PROGRAM pouStation2
VAR
	stationMode: FB_Mode;
	tCalcNumberOfPages: REAL;
	ceil: REAL;
	PartBuild: FB_PartBuild;
	retvall: UDINT;
	// TODO
	tPartPresent: BOOL;
END_VAR

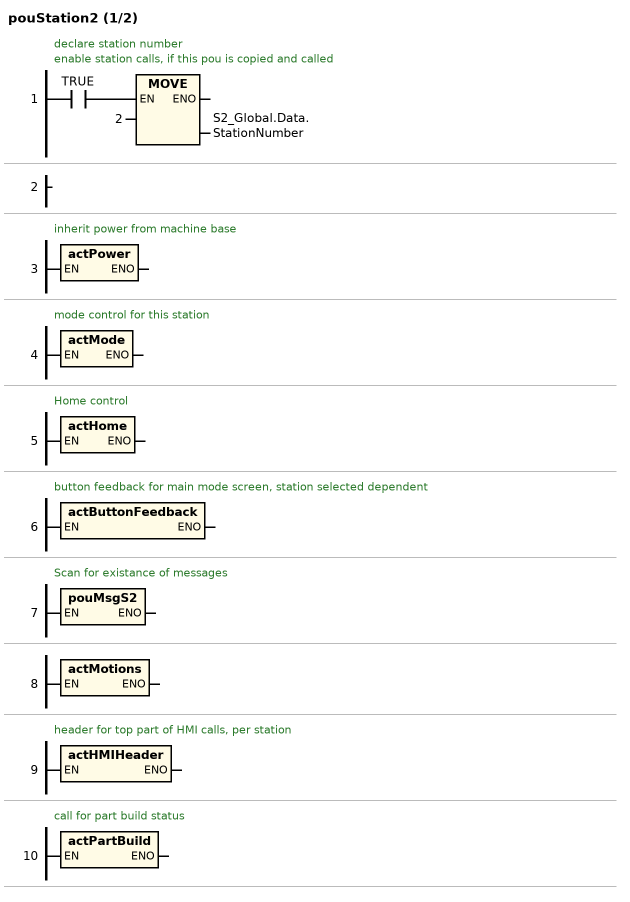
// NETWORK 1
// declare station number
// enable station calls, if this pou is copied and called
S2_Global.Data.StationNumber := 2;

// NETWORK 2

// NETWORK 3
// inherit power from machine base
actPower();

// NETWORK 4
// mode control for this station
actMode();

// NETWORK 5
// Home control
actHome();

// NETWORK 6
// button feedback for main mode screen, station selected dependent
actButtonFeedback();

// NETWORK 7
// Scan for existance of messages
pouMsgS2();

// NETWORK 8
actMotions();

// NETWORK 9
// header for top part of HMI calls, per station
actHMIHeader();

// NETWORK 10
// call for part build status
actPartBuild();

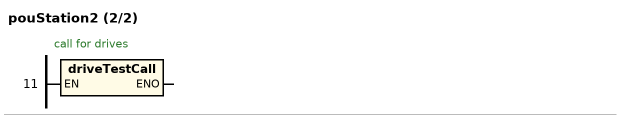
// NETWORK 11
// call for drives
driveTestCall();

ACTION actButtonFeedback:
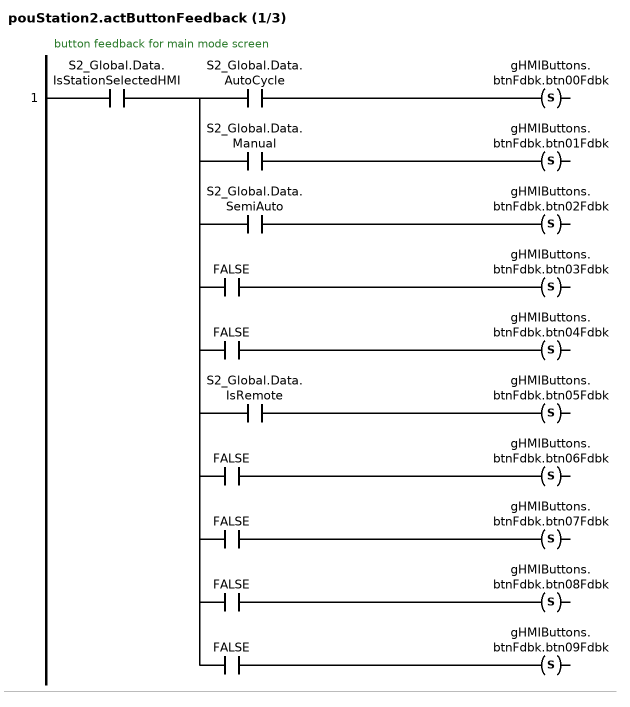
// NETWORK 1
// button feedback for main mode screen
gHMIButtons.btnFdbk.btn00Fdbk S= S2_Global.Data.IsStationSelectedHMI AND S2_Global.Data.AutoCycle;
gHMIButtons.btnFdbk.btn01Fdbk S= S2_Global.Data.IsStationSelectedHMI AND S2_Global.Data.Manual;
gHMIButtons.btnFdbk.btn02Fdbk S= S2_Global.Data.IsStationSelectedHMI AND S2_Global.Data.SemiAuto;
gHMIButtons.btnFdbk.btn03Fdbk S= S2_Global.Data.IsStationSelectedHMI AND FALSE;
gHMIButtons.btnFdbk.btn04Fdbk S= S2_Global.Data.IsStationSelectedHMI AND FALSE;
gHMIButtons.btnFdbk.btn05Fdbk S= S2_Global.Data.IsStationSelectedHMI AND S2_Global.Data.IsRemote;
gHMIButtons.btnFdbk.btn06Fdbk S= S2_Global.Data.IsStationSelectedHMI AND FALSE;
gHMIButtons.btnFdbk.btn07Fdbk S= S2_Global.Data.IsStationSelectedHMI AND FALSE;
gHMIButtons.btnFdbk.btn08Fdbk S= S2_Global.Data.IsStationSelectedHMI AND FALSE;
gHMIButtons.btnFdbk.btn09Fdbk S= S2_Global.Data.IsStationSelectedHMI AND FALSE;

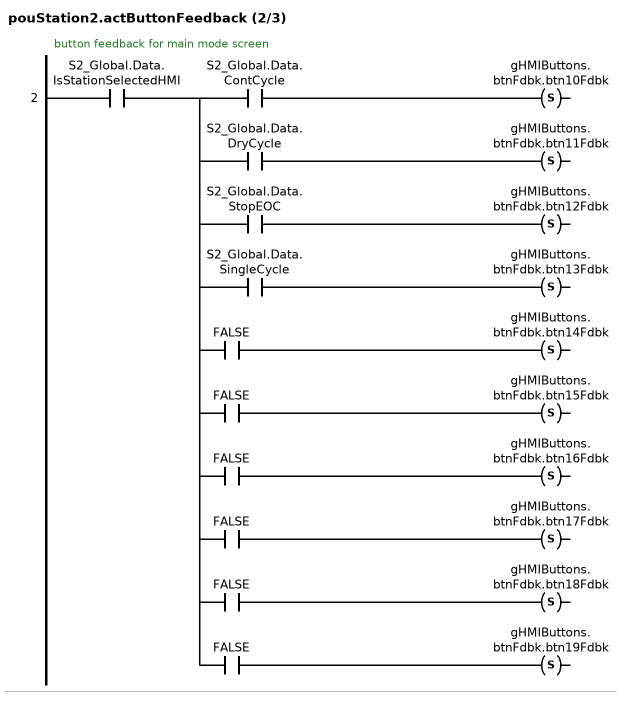
// NETWORK 2
// button feedback for main mode screen
gHMIButtons.btnFdbk.btn10Fdbk S= S2_Global.Data.IsStationSelectedHMI AND S2_Global.Data.ContCycle;
gHMIButtons.btnFdbk.btn11Fdbk S= S2_Global.Data.IsStationSelectedHMI AND S2_Global.Data.DryCycle;
gHMIButtons.btnFdbk.btn12Fdbk S= S2_Global.Data.IsStationSelectedHMI AND S2_Global.Data.StopEOC;
gHMIButtons.btnFdbk.btn13Fdbk S= S2_Global.Data.IsStationSelectedHMI AND S2_Global.Data.SingleCycle;
gHMIButtons.btnFdbk.btn14Fdbk S= S2_Global.Data.IsStationSelectedHMI AND FALSE;
gHMIButtons.btnFdbk.btn15Fdbk S= S2_Global.Data.IsStationSelectedHMI AND FALSE;
gHMIButtons.btnFdbk.btn16Fdbk S= S2_Global.Data.IsStationSelectedHMI AND FALSE;
gHMIButtons.btnFdbk.btn17Fdbk S= S2_Global.Data.IsStationSelectedHMI AND FALSE;
gHMIButtons.btnFdbk.btn18Fdbk S= S2_Global.Data.IsStationSelectedHMI AND FALSE;
gHMIButtons.btnFdbk.btn19Fdbk S= S2_Global.Data.IsStationSelectedHMI AND FALSE;

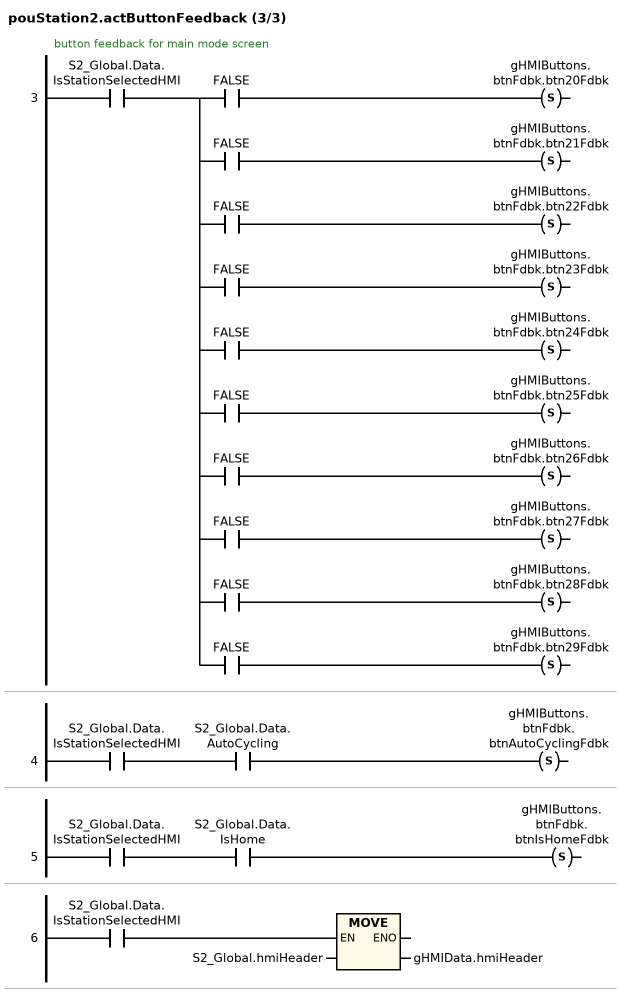
// NETWORK 3
// button feedback for main mode screen
gHMIButtons.btnFdbk.btn20Fdbk S= S2_Global.Data.IsStationSelectedHMI AND FALSE;
gHMIButtons.btnFdbk.btn21Fdbk S= S2_Global.Data.IsStationSelectedHMI AND FALSE;
gHMIButtons.btnFdbk.btn22Fdbk S= S2_Global.Data.IsStationSelectedHMI AND FALSE;
gHMIButtons.btnFdbk.btn23Fdbk S= S2_Global.Data.IsStationSelectedHMI AND FALSE;
gHMIButtons.btnFdbk.btn24Fdbk S= S2_Global.Data.IsStationSelectedHMI AND FALSE;
gHMIButtons.btnFdbk.btn25Fdbk S= S2_Global.Data.IsStationSelectedHMI AND FALSE;
gHMIButtons.btnFdbk.btn26Fdbk S= S2_Global.Data.IsStationSelectedHMI AND FALSE;
gHMIButtons.btnFdbk.btn27Fdbk S= S2_Global.Data.IsStationSelectedHMI AND FALSE;
gHMIButtons.btnFdbk.btn28Fdbk S= S2_Global.Data.IsStationSelectedHMI AND FALSE;
gHMIButtons.btnFdbk.btn29Fdbk S= S2_Global.Data.IsStationSelectedHMI AND FALSE;

// NETWORK 4
gHMIButtons.btnFdbk.btnAutoCyclingFdbk S= S2_Global.Data.IsStationSelectedHMI AND S2_Global.Data.AutoCycling;

// NETWORK 5
gHMIButtons.btnFdbk.btnIsHomeFdbk S= S2_Global.Data.IsStationSelectedHMI AND S2_Global.Data.IsHome;

// NETWORK 6
IF S2_Global.Data.IsStationSelectedHMI THEN gHMIData.hmiHeader := S2_Global.hmiHeader; END_IF
END_ACTION

ACTION actHMIHeader:
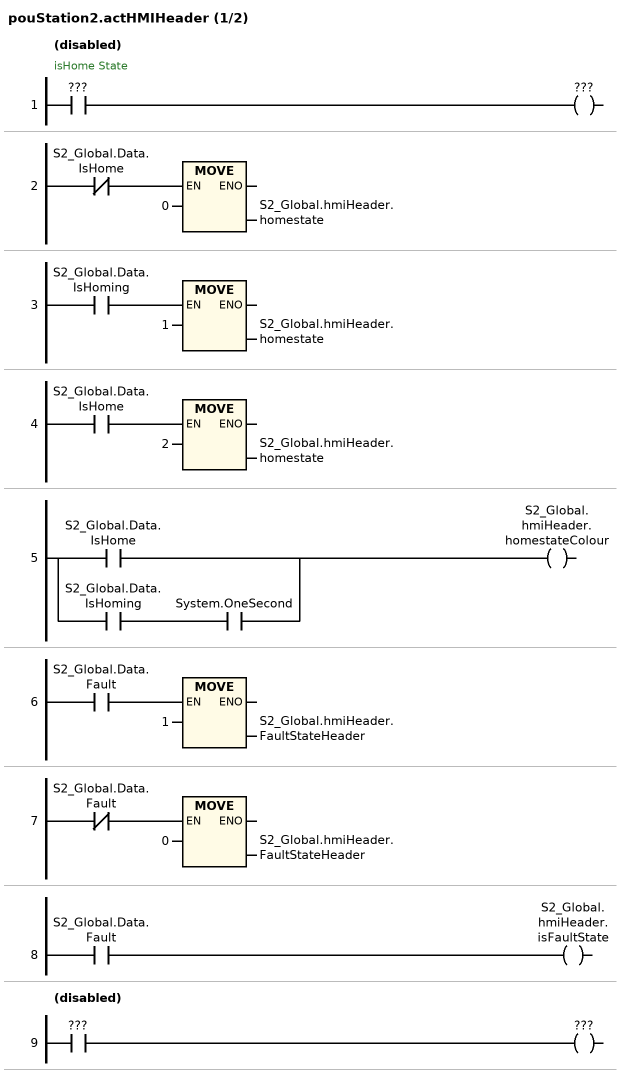
// NETWORK 1 (disabled)
// isHome State
// ??? := ???;

// NETWORK 2
IF NOT S2_Global.Data.IsHome THEN S2_Global.hmiHeader.homestate := 0; END_IF

// NETWORK 3
IF S2_Global.Data.IsHoming THEN S2_Global.hmiHeader.homestate := 1; END_IF

// NETWORK 4
IF S2_Global.Data.IsHome THEN S2_Global.hmiHeader.homestate := 2; END_IF

// NETWORK 5
S2_Global.hmiHeader.homestateColour := S2_Global.Data.IsHome OR S2_Global.Data.IsHoming AND System.OneSecond;

// NETWORK 6
IF S2_Global.Data.Fault THEN S2_Global.hmiHeader.FaultStateHeader := 1; END_IF

// NETWORK 7
IF NOT S2_Global.Data.Fault THEN S2_Global.hmiHeader.FaultStateHeader := 0; END_IF

// NETWORK 8
S2_Global.hmiHeader.isFaultState := S2_Global.Data.Fault;

// NETWORK 9 (disabled)
// ??? := ???;

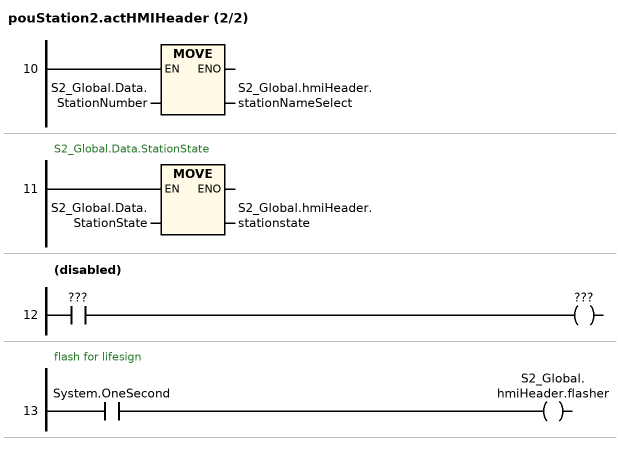
// NETWORK 10
S2_Global.hmiHeader.stationNameSelect := S2_Global.Data.StationNumber;

// NETWORK 11
// S2_Global.Data.StationState
S2_Global.hmiHeader.stationstate := S2_Global.Data.StationState;

// NETWORK 12 (disabled)
// ??? := ???;

// NETWORK 13
// flash for lifesign
S2_Global.hmiHeader.flasher := System.OneSecond;
END_ACTION

ACTION actHome:
//Set home status for station

IF 
//are all motions returned
S2_01_Motion_01_01.Motion.qReturnDepth AND
S2_01_Motion_01_02.Motion.qReturnDepth AND
S2_01_Motion_01_03.Motion.qReturnDepth AND
S2_01_Motion_01_04.Motion.qReturnDepth AND
S2_01_Motion_01_05.Motion.qReturnDepth AND
S2_01_Motion_01_06.Motion.qReturnDepth

	THEN
		//set IsHome value for station
		S2_Global.Data.IsHome := TRUE;
	ELSE
		S2_Global.Data.IsHome := FALSE;
END_IF
END_ACTION

ACTION actMaxNumStationPages:
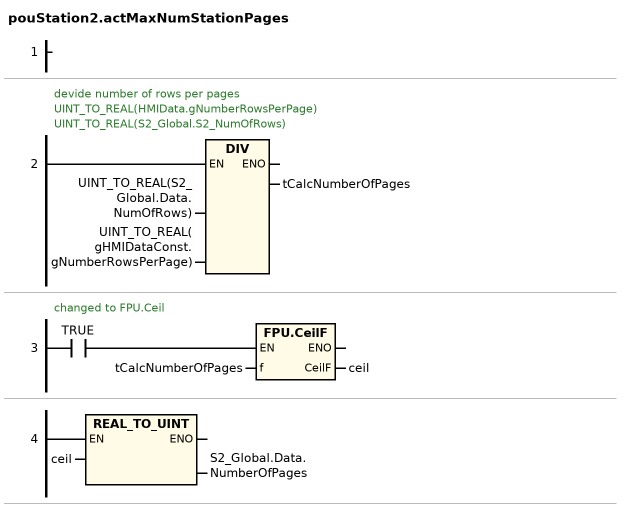
// NETWORK 1

// NETWORK 2
// devide number of rows per pages
// UINT_TO_REAL(HMIData.gNumberRowsPerPage)
// UINT_TO_REAL(S2_Global.S2_NumOfRows)
tCalcNumberOfPages := (UINT_TO_REAL(S2_Global.Data.NumOfRows)) / (UINT_TO_REAL(gHMIDataConst.gNumberRowsPerPage));

// NETWORK 3
// changed to FPU.Ceil
ceil := FPU.CeilF(f := tCalcNumberOfPages);

// NETWORK 4
S2_Global.Data.NumberOfPages := REAL_TO_UINT(ceil);
END_ACTION

ACTION actMode:
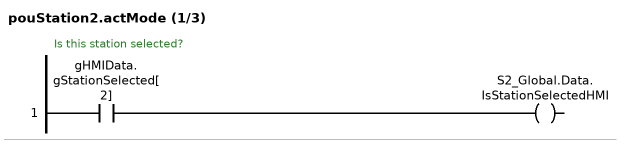
// NETWORK 1
// Is this station selected?
S2_Global.Data.IsStationSelectedHMI := gHMIData.gStationSelected[2];

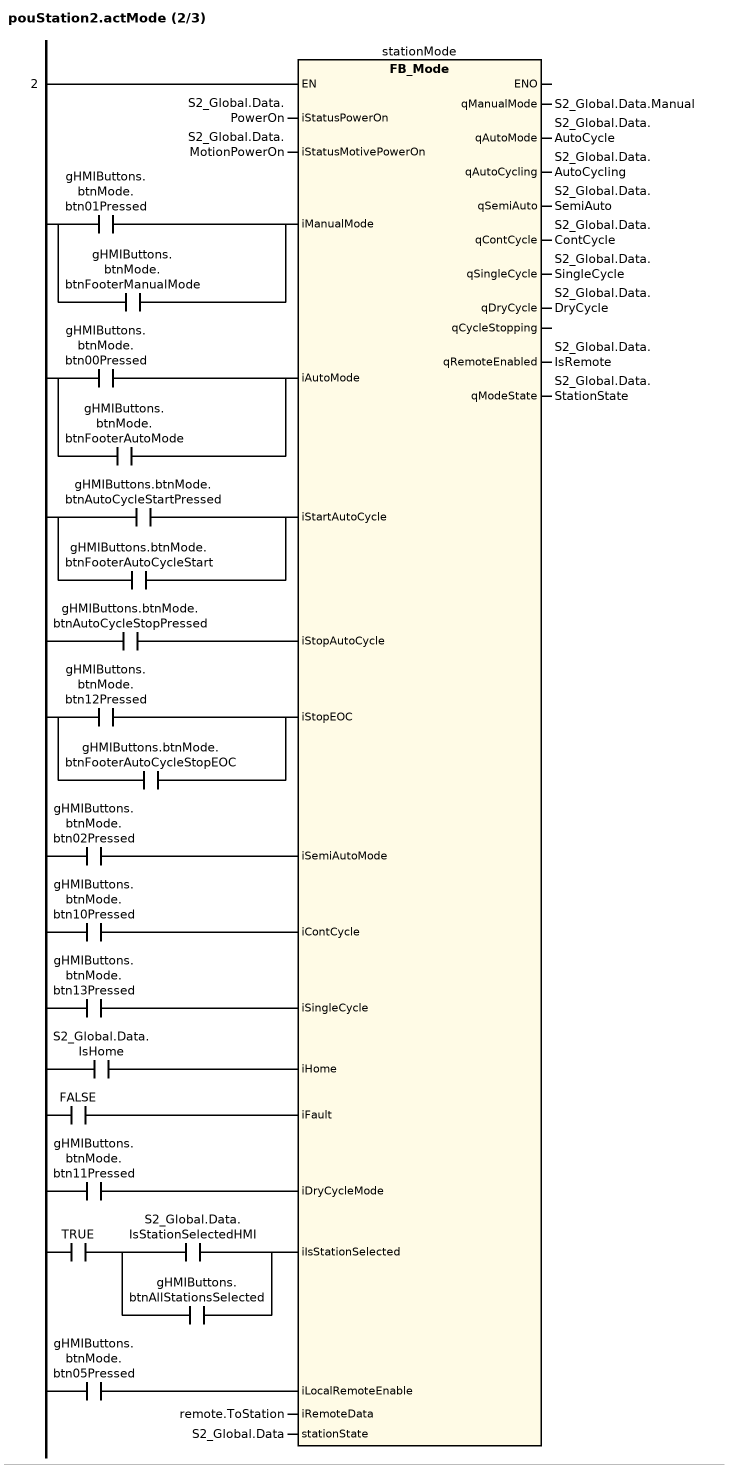
// NETWORK 2
stationMode(
    iStatusPowerOn := S2_Global.Data.PowerOn,
    iStatusMotivePowerOn := S2_Global.Data.MotionPowerOn,
    iManualMode := gHMIButtons.btnMode.btn01Pressed OR gHMIButtons.btnMode.btnFooterManualMode,
    iAutoMode := gHMIButtons.btnMode.btn00Pressed OR gHMIButtons.btnMode.btnFooterAutoMode,
    iStartAutoCycle := gHMIButtons.btnMode.btnAutoCycleStartPressed OR gHMIButtons.btnMode.btnFooterAutoCycleStart,
    iStopAutoCycle := gHMIButtons.btnMode.btnAutoCycleStopPressed,
    iStopEOC := gHMIButtons.btnMode.btn12Pressed OR gHMIButtons.btnMode.btnFooterAutoCycleStopEOC,
    iSemiAutoMode := gHMIButtons.btnMode.btn02Pressed,
    iContCycle := gHMIButtons.btnMode.btn10Pressed,
    iSingleCycle := gHMIButtons.btnMode.btn13Pressed,
    iHome := S2_Global.Data.IsHome,
    iFault := FALSE,
    iDryCycleMode := gHMIButtons.btnMode.btn11Pressed,
    iIsStationSelected := TRUE AND (S2_Global.Data.IsStationSelectedHMI OR gHMIButtons.btnAllStationsSelected),
    iLocalRemoteEnable := gHMIButtons.btnMode.btn05Pressed,
    iRemoteData := remote.ToStation,
    stationState := S2_Global.Data,
    qManualMode => S2_Global.Data.Manual,
    qAutoMode => S2_Global.Data.AutoCycle,
    qAutoCycling => S2_Global.Data.AutoCycling,
    qSemiAuto => S2_Global.Data.SemiAuto,
    qContCycle => S2_Global.Data.ContCycle,
    qSingleCycle => S2_Global.Data.SingleCycle,
    qDryCycle => S2_Global.Data.DryCycle,
    qRemoteEnabled => S2_Global.Data.IsRemote,
    qModeState => S2_Global.Data.StationState); // FB_Mode

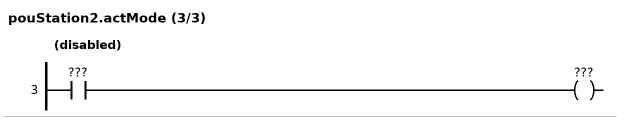
// NETWORK 3 (disabled)
// ??? := ???;
END_ACTION

ACTION actMotions:
//station 1 = 10000 index


//init number of rows
S2_Global.Data.NumOfRows := 0;

//page 1
S2_01_Motion_01_01();
S2_01_Motion_01_02();
S2_01_Motion_01_03();
S2_01_Motion_01_04();
S2_01_Motion_01_05();
S2_01_Motion_01_06();

//page 2
S2_01_Motion_02_07();
S2_01_Motion_02_08();
S2_01_Motion_02_09();
S2_01_Motion_02_10();
S2_01_Motion_02_11();
S2_01_Motion_02_12();

//page 3
S2_01_Motion_03_13();
S2_01_Motion_03_14();
S2_01_Motion_03_15();
S2_01_Motion_03_16();
S2_01_Motion_03_17();
S2_01_Motion_03_18();

//page 4
S2_01_Motion_04_19();
S2_01_Motion_04_20();
S2_01_Motion_04_21();
S2_01_Motion_04_22();
S2_01_Motion_04_23();
S2_01_Motion_04_24();

//page 5
S2_01_Motion_05_25();
S2_01_Motion_05_26();
S2_01_Motion_05_27();
S2_01_Motion_05_28();
S2_01_Motion_05_29();
S2_01_Motion_05_30();

//page 6
S2_01_Motion_06_31();
S2_01_Motion_06_32();
S2_01_Motion_06_33();
S2_01_Motion_06_34();
S2_01_Motion_06_35();
S2_01_Motion_06_36();

//must be called after motionRow calls
actMaxNumStationPages();
END_ACTION

ACTION actPartBuild:
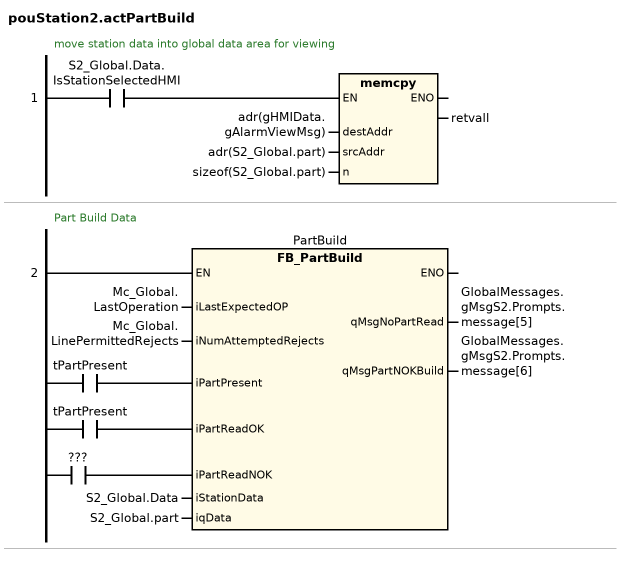
// NETWORK 1
// move station data into global data area for viewing
IF S2_Global.Data.IsStationSelectedHMI THEN
    retvall := memcpy(destAddr := adr(gHMIData.gAlarmViewMsg), srcAddr := adr(S2_Global.part), n := sizeof(S2_Global.part));
END_IF

// NETWORK 2
// Part Build Data
PartBuild(
    iLastExpectedOP := Mc_Global.LastOperation,
    iNumAttemptedRejects := Mc_Global.LinePermittedRejects,
    iPartPresent := tPartPresent,
    iPartReadOK := tPartPresent,
    iStationData := S2_Global.Data,
    iqData := S2_Global.part,
    qMsgNoPartRead => GlobalMessages.gMsgS2.Prompts.message[5],
    qMsgPartNOKBuild => GlobalMessages.gMsgS2.Prompts.message[6]); // FB_PartBuild
END_ACTION

ACTION actPower:
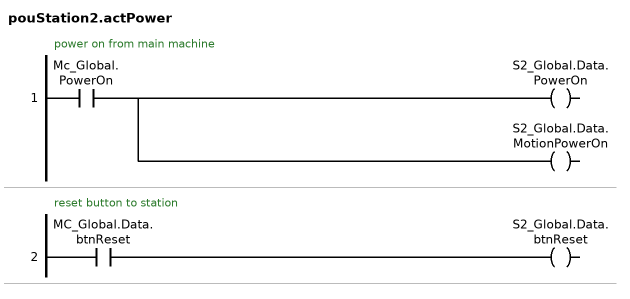
// NETWORK 1
// power on from main machine
S2_Global.Data.PowerOn := Mc_Global.PowerOn;
S2_Global.Data.MotionPowerOn := Mc_Global.PowerOn;

// NETWORK 2
// reset button to station
S2_Global.Data.btnReset := MC_Global.Data.btnReset;
END_ACTION

END_PROGRAM

(* stored: Version 1.1.0.1, ProductVersion 3.1.4024.12
   POU pouStation2: Id {fd8ca611-dcd7-4808-b220-3ca7fa511e9d}, SpecialFunc None
   Action actButtonFeedback: Id {53e81109-c13a-4493-b591-48fbf4002db6}
   Action actHMIHeader: Id {ee50a15d-d766-4744-a0fd-ffe9c4f8646c}
   Action actHome: Id {0883900f-8058-40f6-a4c3-fae5254b2ba8}
   Action actMaxNumStationPages: Id {7ce2426d-b6e4-45d9-acfd-953f5fdcae61}
   Action actMode: Id {89491c54-f09e-4480-a81d-ba1f3bfa5019}
   Action actMotions: Id {66fa6756-b646-460a-b835-0014fc22e25b}
   Action actPartBuild: Id {f0f8c37e-cd13-490d-a003-cb5f08cd140b}
   Action actPower: Id {7bbc8cd9-3e8d-40ea-83fb-9a607850df83} *)
